// TIA Portal V18 export
VAR_GLOBAL   // PLC tag table "默认变量表"
   Tag_1 AT %M0.0 : Bool;
   Tag_2 AT %M0.1 : Bool;
   Tag_3 AT %M1.1 : Bool;
   Tag_4 AT %M1.2 : Bool;
END_VAR
